// TIA Portal V18 export
TYPE "UDT_settings"
   STRUCT
      taktTimeCntOption { ExternalVisible := 'False'; S7_SetPoint := 'True'} : DInt;   // 0: off / 1: manual / automatic
      target { ExternalVisible := 'False'; S7_SetPoint := 'True'} : DInt;   // Target production pcs
      taktTime { ExternalVisible := 'False'; S7_SetPoint := 'True'} : DInt;   // Takt time in ms
      countOption { ExternalVisible := 'False'; S7_SetPoint := 'True'} : DInt;   // 0: ?? / 1: ??
      shiftTargetEn { ExternalVisible := 'False'; S7_SetPoint := 'True'} : DInt;
      shiftTaktTimeEn { ExternalVisible := 'False'; S7_SetPoint := 'True'} : DInt;
   END_STRUCT;
END_TYPE
